TYPE ST_OperatorAct :
STRUCT
	Batch		: STRING(100);
	DateTime	: DT;
	Event		: STRING(100);
	Description	: STRING(100);
END_STRUCT
END_TYPE

(* stored: Version 1.1.0.1, ProductVersion 3.1.4024.12
   DUT ST_OperatorAct: Id {85b9304d-dd3b-4ba7-9e37-0071db8283a1} *)
